// TIA Portal V19 export
DATA_BLOCK "A03_HMI_IDB"   // DB72
AUTHOR : Piemme
FAMILY : System
// stored: InstanceOfName HMI_A03_FB, InstanceOfType FB
"HMI_A03_FB"
   // VAR_OUTPUT
   //    MB3_LpJog : Bool;
   // END_VAR
   // VAR
   //    MB3_Decoder { ExternalAccessible := 'False'; ExternalVisible := 'False'; ExternalWritable := 'False'} : "ButtonsHMIDecoder";
   // END_VAR
BEGIN
END_DATA_BLOCK
